PROGRAM MAIN
VAR
END_VAR

// Niet gemaakt

(*
Druktoets functies

Maak een FB DrukknopSpecial aan die een drukknop speciale functies geeft zoals

    Één enkele klik
    Dubbele klik
    Lang klikken ( > 1s )

Dit zijn natuurlijk drie aparte uitgangen en slechts één ingang.
*)

END_PROGRAM

(* stored: Version 1.1.0.1, ProductVersion 3.1.4024.12
   POU MAIN: Id {c43055ab-c7f9-4244-8b31-5d4dbf71b705}, SpecialFunc None *)
